PROGRAM MAIN
VAR
	fbAxisStMachine : FB_AxisStMachineMaster;
END_VAR

fbAxisStMachine(AxisInOut := GVL.Axis_Virtual);

END_PROGRAM

(* stored: Version 1.1.0.1, ProductVersion 3.1.4024.12
   POU MAIN: Id {820171f7-8670-42df-9df1-221fdd638619}, SpecialFunc None *)
